(* CoDeSys 2.3.9.22 project: pr2.pro *)
(* Libraries: Util.lib 18.5.10 15:14:28, STANDARD.LIB 4.10.05 11:14:46, IECSFC.LIB 13.4.06 15:51:28 *)

(* PLC configuration (modules and I/O channels)
start AT %IX0.0 [BitInput]
continue AT %IX0.1 [BitInput]
stop AT %IX0.2 [BitInput]
AT %IX0.3 [BitInput]
AT %IX0.4 [BitInput]
AT %IX0.5 [BitInput]
Discrete output 4 bit [ID101] node 1, in %IB1 out %QB1 {PinCount = 4; SafeValueBool = FALSE; SafeValueBool = FALSE; SafeValueBool = FALSE; SafeValueBool = FALSE; Visibility = No}
  AT %QX1.0 [BitOutput]
  AT %QX1.1 [BitOutput]
  AT %QX1.2 [BitOutput]
  AT %QX1.3 [BitOutput]
Special output [ID104] node 2, in %IB2 out %QB2 {Visibility = No; PinCount = 1}
  AT %QX2.0 [BitOutput] Special output
Unifed signal sensor [ID700] node 3, in %IB3 out %QB3 {Type_of_sensor700 = IT_0_20; measure_interval = 0.8; ainlow = 0; ainhigh = 20; first_cor_point = 0; first_delta = 0; second_cor_point = 0; second_delta = 0; third_cor_point = 0; third_delta = 0; Visibility = No}
  AT %ID3.0 [FloatInput] Value
  AT %IW3.1 [WordInput] Circular time
  Analog Input [ID107] node 0, in %IB3.0 out %QB3.0
Unifed signal sensor [ID700] node 4, in %IB4 out %QB4 {Type_of_sensor700 = IT_0_20; measure_interval = 0.8; ainlow = 0; ainhigh = 20; first_cor_point = 0; first_delta = 0; second_cor_point = 0; second_delta = 0; third_cor_point = 0; third_delta = 0; Visibility = No}
  AT %ID4.0 [FloatInput] Value
  AT %IW4.1 [WordInput] Circular time
  Analog Input [ID107] node 0, in %IB4.0 out %QB4.0
Unifed signal sensor [ID700] node 5, in %IB5 out %QB5 {Type_of_sensor700 = IT_0_20; measure_interval = 0.8; ainlow = 0; ainhigh = 20; first_cor_point = 0; first_delta = 0; second_cor_point = 0; second_delta = 0; third_cor_point = 0; third_delta = 0; Visibility = No}
  AT %ID5.0 [FloatInput] Value
  AT %IW5.1 [WordInput] Circular time
  Analog Input [ID107] node 0, in %IB5.0 out %QB5.0
Unifed signal sensor [ID700] node 6, in %IB6 out %QB6 {Type_of_sensor700 = IT_0_20; measure_interval = 0.8; ainlow = 0; ainhigh = 20; first_cor_point = 0; first_delta = 0; second_cor_point = 0; second_delta = 0; third_cor_point = 0; third_delta = 0; Visibility = No}
  AT %ID6.0 [FloatInput] Value
  AT %IW6.1 [WordInput] Circular time
  Analog Input [ID107] node 0, in %IB6.0 out %QB6.0
Analog output [ID106] node 7, in %IB7 out %QB7 {DAC_Type = Current 4-20mA; Analog_offset_correction = 0; Analog_full_range_correction = 0; SafeValueFloat = 0; Visibility = No}
  AT %QD7.0 [FloatOutput] Value
Analog output [ID106] node 8, in %IB8 out %QB8 {DAC_Type = Current 4-20mA; Analog_offset_correction = 0; Analog_full_range_correction = 0; SafeValueFloat = 0; Visibility = No}
  AT %QD8.0 [FloatOutput] Value
*)

(* POU PLC_PRG, CFC *)
PROGRAM PLC_PRG
VAR
	rs1: RS;
	Y1: REAL;
	ton1: TON;
	ton2: TON;
	on: BOOL;
	X1: REAL;
	ton3: TON;
	blink1: BLINK;
	cv1: REAL;
	ctu1: CTU;
	bar: BOOL;
	ton4: TON;
	rs2: RS;
	ton5: TON;
	ton6: TON;
	blink2: BLINK;
	vent: BOOL;
	ton7: TON;
	ton8: TON;
	rs3: RS;
	ton9: TON;
	endC: BOOL;
	rs4: RS;
	bkink3: BLINK;
	rs5: RS;
	KB: BOOL;
	P3: BOOL;
	PC: BOOL;

	stopOFF: BOOL;
	blink4: BLINK;
	blinkOFF: BOOL;
	vanish: BOOL;
	rotate: REAL := 0;
	ctuRot: CTU;
	viz1: BOOL;
	viz2: BOOL;
END_VAR
VAR (* helpers for the ST form of the networks *)
	_t485 : BOOL;
	_t571 : BOOL;
	_t515 : BOOL;
	_t479 : BOOL;
	_t526 : BOOL;
	_t445 : BOOL;
	_t432 : REAL;
	_t450 : REAL;
	_t473 : REAL;
	_t474 : REAL;
	_t472 : REAL;
	_t545 : BOOL;
	_t583 : BOOL;
END_VAR
_CFC_ (* Continuous Function Chart, elements in execution order *)
#0 rs5:RS(SET: #21, RESET1: #18.Q)
#1 R bar <= #32.Q
#2 ton7:TON(IN: #39.Q, PT: T#4s500ms)
#3 EQ(Y1, 2000)
#4 R endC <= #21
#5 R stopOFF <= #21
#6 R blinkOFF <= #21
#7 S on <= start
#8 rs1:RS(SET: #21, RESET1: #54.Q)
#9 ton1:TON(IN: #8.Q1, PT: T#8s)
#10 ton2:TON(IN: #9.Q, PT: T#5s)
#11 TIME_TO_REAL(#9.ET)
#12 MUL(#11, -1)
#13 Y1 <= #12
#14 TIME_TO_REAL(#10.ET)
#15 X1 <= #14
#16 ton3:TON(IN: #10.Q, PT: T#10s)
#17 blink1:BLINK(ENABLE: #25, TIMELOW: T#2s, TIMEHIGH: T#2s)
#18 ctu1:CTU(CU: #17.OUT, RESET: #18.Q, PV: 4)
#19 cv1 <= #18.CV
#20 TIME_TO_REAL(#16.ET)
#21 OR(start, #59)
#22 ADD(Y1, #20)
#23 Y1 <= #22
#24 rs2:RS(SET: #18.Q, RESET1: #54.Q)
#25 AND(#16.Q, #0.Q1)
#26 bar <= #37
#27 ton4:TON(IN: #24.Q1, PT: T#10s)
#28 TIME_TO_REAL(#27.ET)
#29 MUL(-1, #28)
#30 ADD(Y1, #29)
#31 Y1 <= #30
#32 ton5:TON(IN: #27.Q, PT: T#3s)
#33 TIME_TO_REAL(#32.ET)
#34 MUL(-1, #33)
#35 ADD(X1, #34)
#36 X1 <= #35
#37 AND(#0.Q1, #17.OUT, #3)
#38 vent <= #45
#39 ton6:TON(IN: #32.Q, PT: T#10s)
#40 ADD(Y1, #44)
#41 Y1 <= #40
#42 AND(#39.Q, NOT #46.Q1)
#43 blink2:BLINK(ENABLE: #42, TIMELOW: T#2s, TIMEHIGH: T#4s)
#44 TIME_TO_REAL(#39.ET)
#45 AND(#43.OUT, NOT #46.Q1)
#46 rs3:RS(SET: #2.Q, RESET1: #54.Q)
#47 ton8:TON(IN: #46.Q1, PT: T#8s)
#48 MUL(-1, #51)
#49 ADD(Y1, #48)
#50 Y1 <= #49
#51 TIME_TO_REAL(#47.ET)
#52 ADD(X1, #55)
#53 bkink3:BLINK(ENABLE: #60.Q1, TIMELOW: T#1s, TIMEHIGH: T#1s)
#54 ton9:TON(IN: #47.Q, PT: T#2s)
#55 MUL(-1, #56)
#56 TIME_TO_REAL(#54.ET)
#57 endC <= #67
#58 X1 <= #52
#59 AND(NOT #54.Q, continue, on)
#60 rs4:RS(SET: #54.Q, RESET1: #59)
#61 EQ(Y1, -8000)
#62 KB <= #61
#63 EQ(X1, 5000)
#64 P3 <= #63
#65 EQ(X1, 2000)
#66 PC <= #65
#67 AND(#53.OUT, #60.Q1, NOT stopOFF, on, #68)
#68 EQ(X1, 0)
#69 R on <= stop
#70 S vanish <= #21
#71 R endC <= stop
#72 S blinkOFF <= stop
#73 S stopOFF <= stop
#74 R vanish <= stop
#75 viz1 <= #76.OUT
#76 blink4:BLINK(ENABLE: #37, TIMELOW: T#0.5s, TIMEHIGH: T#0.5s)
#77 viz2 <= NOT #76.OUT
_END_CFC_
(* the same logic as Structured Text *)
rs5(SET := _t485, RESET1 := ctu1.Q);
IF ton5.Q THEN bar := FALSE; END_IF;
ton7(IN := ton6.Q, PT := T#4s500ms);
_t571 := Y1 = 2000;
IF _t485 THEN endC := FALSE; END_IF;
IF _t485 THEN stopOFF := FALSE; END_IF;
IF _t485 THEN blinkOFF := FALSE; END_IF;
IF start THEN on := TRUE; END_IF;
rs1(SET := _t485, RESET1 := ton9.Q);
ton1(IN := rs1.Q1, PT := T#8s);
ton2(IN := ton1.Q, PT := T#5s);
Y1 := TIME_TO_REAL(ton1.ET) * (-1);
X1 := TIME_TO_REAL(ton2.ET);
ton3(IN := ton2.Q, PT := T#10s);
blink1(ENABLE := _t515, TIMELOW := T#2s, TIMEHIGH := T#2s);
ctu1(CU := blink1.OUT, RESET := ctu1.Q, PV := 4);
cv1 := ctu1.CV;
_t485 := start OR _t479;
Y1 := Y1 + TIME_TO_REAL(ton3.ET);
rs2(SET := ctu1.Q, RESET1 := ton9.Q);
_t515 := ton3.Q AND rs5.Q1;
bar := _t526;
ton4(IN := rs2.Q1, PT := T#10s);
Y1 := Y1 + ((-1) * TIME_TO_REAL(ton4.ET));
ton5(IN := ton4.Q, PT := T#3s);
X1 := X1 + ((-1) * TIME_TO_REAL(ton5.ET));
_t526 := rs5.Q1 AND blink1.OUT AND _t571;
vent := _t445;
ton6(IN := ton5.Q, PT := T#10s);
Y1 := Y1 + _t432;
blink2(ENABLE := ton6.Q AND NOT rs3.Q1, TIMELOW := T#2s, TIMEHIGH := T#4s);
_t432 := TIME_TO_REAL(ton6.ET);
_t445 := blink2.OUT AND NOT rs3.Q1;
rs3(SET := ton7.Q, RESET1 := ton9.Q);
ton8(IN := rs3.Q1, PT := T#8s);
Y1 := Y1 + ((-1) * _t450);
_t450 := TIME_TO_REAL(ton8.ET);
_t474 := X1 + _t473;
bkink3(ENABLE := rs4.Q1, TIMELOW := T#1s, TIMEHIGH := T#1s);
ton9(IN := ton8.Q, PT := T#2s);
_t473 := (-1) * _t472;
_t472 := TIME_TO_REAL(ton9.ET);
endC := _t545;
X1 := _t474;
_t479 := NOT ton9.Q AND continue AND on;
rs4(SET := ton9.Q, RESET1 := _t479);
KB := Y1 = (-8000);
P3 := X1 = 5000;
PC := X1 = 2000;
_t545 := bkink3.OUT AND rs4.Q1 AND NOT stopOFF AND on AND _t583;
_t583 := X1 = 0;
IF stop THEN on := FALSE; END_IF;
IF _t485 THEN vanish := TRUE; END_IF;
IF stop THEN endC := FALSE; END_IF;
IF stop THEN blinkOFF := TRUE; END_IF;
IF stop THEN stopOFF := TRUE; END_IF;
IF stop THEN vanish := FALSE; END_IF;
viz1 := blink4.OUT;
blink4(ENABLE := _t526, TIMELOW := T#0.5s, TIMEHIGH := T#0.5s);
viz2 := NOT blink4.OUT;
END_PROGRAM

(* Visualisation w1
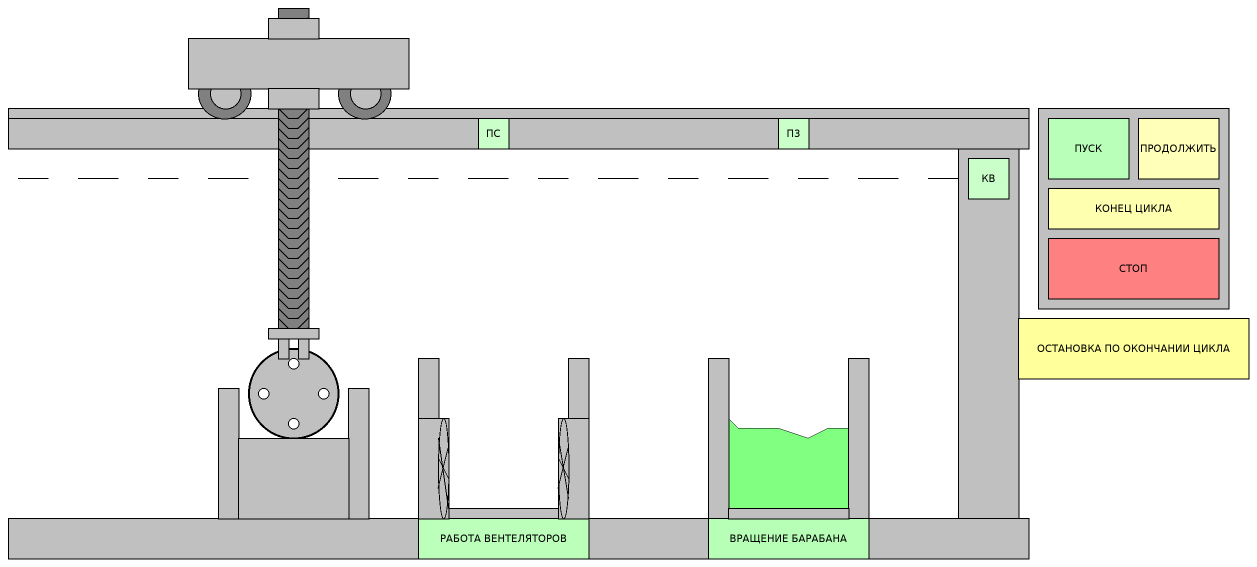
rounded rectangle at (290,550)-(301,581): x offset PLC_PRG.X1/10; y offset PLC_PRG.Y1/50
rounded rectangle at (270,550)-(281,581): x offset PLC_PRG.X1/10; y offset PLC_PRG.Y1/50
rounded rectangle at (1040,340)-(1121,401): text "ПУСК"; alarm colour if PLC_PRG.on; taps .start
rounded rectangle at (960,380)-(1001,421): text "КВ"; alarm colour if PLC_PRG.KB
rectangle at (700,740)-(861,781): text "ВРАЩЕНИЕ БАРАБАНА"; alarm colour if PLC_PRG.bar
rounded rectangle at (770,340)-(801,371): text "П3"; alarm colour if PLC_PRG.P3
rounded rectangle at (470,340)-(501,371): text "ПС"; alarm colour if PLC_PRG.PC
rectangle at (410,740)-(581,781): text "РАБОТА ВЕНТЕЛЯТОРОВ"; alarm colour if PLC_PRG.vent
rectangle at (1040,410)-(1211,451): text "КОНЕЦ ЦИКЛА"; alarm colour if PLC_PRG.endC
rounded rectangle at (1130,340)-(1211,401): text "ПРОДОЛЖИТЬ"; alarm colour if PLC_PRG.endC; taps .continue
rounded rectangle at (260,240)-(311,261): x offset PLC_PRG.X1/10
rounded rectangle at (260,310)-(311,331): x offset PLC_PRG.X1/10
rounded rectangle at (260,550)-(311,561): x offset PLC_PRG.X1/10; y offset PLC_PRG.Y1/50
rounded rectangle at (1040,460)-(1211,521): text "СТОП"; alarm colour if PLC_PRG.stopOFF; taps .stop
rounded rectangle at (1010,540)-(1241,601): text "ОСТАНОВКА ПО ОКОНЧАНИИ ЦИКЛА"; invisible if PLC_PRG.vanish
88 more shapes without text or variables
*)
